{attribute addProperty BoxType "EK1122-0000-0018"}
{attribute addProperty Id "Beckhoff_EL72xxsub_EK1100EK1100_179A0949162"}
{attribute addProperty CRC "3665775472"}
{attribute addProperty SizeInBites "16"}
{attribute addProperty SizeInBytes "2"}
TYPE Beckhoff_EL72xxEK1122_DA7F4B70 EXTENDS EK1122_179A0949 :
STRUCT
	{attribute addProperty Name "Beckhoff_EL72xxsub_EK1100"}
	Beckhoff_EL72xxsub_EK1100 : EK1100_179A0949;
END_STRUCT
END_TYPE

(* stored: Version 1.2.0.0, ProductVersion 3.1.4024.9
   DUT Beckhoff_EL72xxEK1122_DA7F4B70: Id {8aa29dc3-8c66-4a2c-8f06-0d181510975f} *)
